(* CoDeSys 2.3.9.55 project: PuertaGaraje.pro *)
(* Libraries: Standard.lib 2.6.14 10:37:46 *)

(* Global variable list: Global_Variables *)
VAR_GLOBAL

   (* Entradas *)
   P : BOOL;
   FCA:BOOL;
  FCC: BOOL;

   (* Salidas *)
   Abrir: BOOL;
   Cerrar : BOOL;

END_VAR

(* POU PLC_PRG, ST *)
PROGRAM PLC_PRG
VAR
END_VAR
Animacion();
ControlLD();
END_PROGRAM

(* POU Animacion, ST *)
PROGRAM Animacion
VAR
    Pos : INT;
END_VAR
IF (Abrir AND Pos>-160) THEN
   Pos:=Pos-3;
END_IF

IF (Cerrar AND POS<0) THEN
   Pos:=Pos+3;
END_IF

FCC:= (Pos>=0) ;
FCA:=(Pos<=-160);
END_PROGRAM

(* POU ControlLD, LD *)
PROGRAM ControlLD
VAR

END_VAR
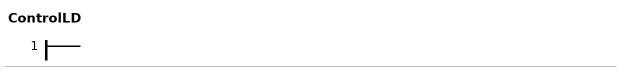
_LD_ (* Ladder Diagram *)
NETWORK 1
	*
_END_LD_
(* the same logic as Structured Text *)
(* Network 1 *)
END_PROGRAM

(* Visualisation Visu
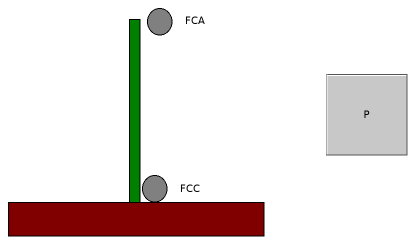
button at (450,140)-(531,221): text "P"; taps P
rectangle at (253,85)-(264,269): bottom Animacion.Pos
ellipse at (266,241)-(291,268): alarm colour if FCC
ellipse at (271,74)-(296,101): alarm colour if FCA
rectangle at (286,244)-(342,265): text "FCC"
rectangle at (291,76)-(347,97): text "FCA"
1 more shapes without text or variables
*)
